(* PLC project agitator_1speed, Dassault Systèmes ControlBuild 2024x *)
(* stored: creationDateTime 2023-10-03T11:13:03-01:00 *)

(* This module simulates the behaviour of a 1-speed motorized agitator and its electrical control logic. *)
FUNCTION_BLOCK equipment_library.agitator_1speed
  VAR_INPUT
    voltage380 : BOOL := true;
    cmdSupply : BOOL := true;
    sensorSupply : BOOL := true;
  END_VAR
  VAR_INPUT
    cmd : BOOL := false;
  END_VAR
  VAR_OUTPUT
    cmdFB : BOOL := false;
    thermal : BOOL := false;
  END_VAR
  VAR_OUTPUT
    speedVal : REAL := 0.0;
    speedPercent : REAL := 0.0;
  END_VAR
  VAR
    increment : REAL := 0.0;
    memo : BOOL := false;
    state : BOOL := false;
    speedSetpoint : REAL := 0.0;
    cnt : DINT := 0;
    flipflop : BOOL := false;
  END_VAR
  VAR CONSTANT
    nominalTime : REAL := 0.5;
    thermalLogic : BOOL := false;
    cmdFbLogic : BOOL := true;
    nominalSpeed : REAL := 5000.0;
  END_VAR
  VAR
    d_locking : BOOL := false;
    v_d_locking : REAL := 0.0;
    d_electrical : BOOL := false;
    v_d_electrical : BOOL := false;
    d_cmdFB : BOOL := false;
    v_d_cmdFB : BOOL := false;
  END_VAR


ACTION C_source_code:
/* -----------------------------------------------------------------	*/
/* Type : Model of Operative Behaviour					*/
/* Catégorie :   batch							*/
/* Author : Dassault Systemes						*/
/* Update date : June 2018							*/
/* -----------------------------------------------------------------	*/
/* This module simulates the behaviour of a 1-speed motorized		*/
/* agitator and its electrical control logic.				*/
/* ----------------------------------------------------------------	*/

/* ----------------------------------------------------------------	*/
/* Management of orders from Control Part					*/
/*	if there is no power supply for command 				*/
/*     the contactor doesn't understand the control order		*/
/* ----------------------------------------------------------------	*/
if (cmd && cmdSupply) memo = 1;
if (!cmd || !cmdSupply || d_electrical) memo = 0;

/* ----------------------------------------------------------------	*/
/* Calculation of the on-state of contactor				*/
/* ----------------------------------------------------------------	*/
state=memo & voltage380;

/* ----------------------------------------------------------------	*/
/* Management of the speed ramp						*/
/* ----------------------------------------------------------------	*/
if (d_locking)  speedVal = v_d_locking;
else {
	/* Compute the speed setpoint according to contator's state	*/
	speedSetpoint = 0.0;
	if (state) {
		speedSetpoint = nominalSpeed;
		if (nominalTime > 0.0)
			increment = (nominalSpeed / nominalTime) * (CLOCK_PERIOD/1000000.0);
	}

	/* Compute the speed ramp	*/
	if ( speedVal < speedSetpoint ) {
		speedVal += increment;
		if ( speedVal > speedSetpoint ) speedVal = speedSetpoint;
	}
	if ( speedVal > speedSetpoint ) {
		speedVal -= increment;
		if (speedVal < speedSetpoint) speedVal = speedSetpoint;
	}
}

/* ----------------------------------------------------------------	*/
/* Compute the percentage between the current and nominal speed	*/
/* ----------------------------------------------------------------	*/
if (nominalSpeed != 0.0)
	speedPercent = ((speedVal/nominalSpeed)*100);

/* ----------------------------------------------------------------	*/
/* Management of the thermal feedback					*/
/* ----------------------------------------------------------------	*/
if (d_electrical) thermal=v_d_electrical;
else
	thermal= ! thermalLogic && sensorSupply;

/* ----------------------------------------------------------------	*/
/* Management of feedback to Control Part					*/
/*     if a fault is required, the contactor feed-back 		*/
/*		 takes a preset state.					*/
/*	if there is no power supply for sensors 				*/
/*         contactor feed-back returns nothing				*/
/*     else contactor feed-back returns the contactor state combined	*/
/*	    with wiring logic.						*/
/* ----------------------------------------------------------------	*/
if (d_cmdFB) cmdFB = v_d_cmdFB;
else 	
	cmdFB = (memo ^ ! cmdFbLogic) && sensorSupply;

/* ----------------------------------------------------------------	*/
/* Animation of blades : only for MAN					*/
/* ----------------------------------------------------------------	*/
if (speedPercent != 0.0) {
	if (! flipflop) cnt ++;
	else cnt --;
	if (cnt >4) {
		cnt = 4;
		flipflop = 1;
	}
	if (cnt <= 0) flipflop = 0;
}
END_ACTION
END_FUNCTION_BLOCK
